{attribute 'GeneratedUsingTerminal: EK1200-1388-0000'}
{attribute addProperty BoxType "EK1200-1388-0000"}
{attribute addProperty Id "Term_2_EL6002EL6002_81703A53126Term_3_EL1809EL1809_32157CFD20Term_4_EL2809EL2809_2B6483BD19Term_5_EL4004EL4004_D2A7C9B719Term_6_EL2809EL2809_2B6483BD19Term_7_EL6001EL6001_B592E1CA69"}
{attribute addProperty CRC "875215620"}
{attribute addProperty Size "272"}
TYPE Term_1_EK1200_342ABB04 :
STRUCT
	{attribute addProperty Name "Term_2_EL6002"}
	Term_2_EL6002 : EL6002_81703A53;
	{attribute addProperty Name "Term_3_EL1809"}
	Term_3_EL1809 : EL1809_32157CFD;
	{attribute addProperty Name "Term_4_EL2809"}
	Term_4_EL2809 : EL2809_2B6483BD;
	{attribute addProperty Name "Term_5_EL4004"}
	Term_5_EL4004 : EL4004_D2A7C9B7;
	{attribute addProperty Name "Term_6_EL2809"}
	Term_6_EL2809 : EL2809_2B6483BD;
	{attribute addProperty Name "Term_7_EL6001"}
	Term_7_EL6001 : EL6001_B592E1CA;
END_STRUCT
END_TYPE

(* stored: Version 1.2.0.0, ProductVersion 3.1.4024.9
   DUT Term_1_EK1200_342ABB04: Id {f4cae944-f2a3-0962-0e14-e0064bd77fc5} *)
